(* CoDeSys 2.3 export: INDICATOR_CTRL.EXP *)

(* POU lib/INDICATOR_CTRL, FBD *)
FUNCTION_BLOCK INDICATOR_CTRL
VAR_INPUT
	iSTATE						:	INT;
	xEMERGENCY			:	BOOL;
	xRUNNING				:	BOOL;
	xCLOCK					:	BOOL;
END_VAR
VAR_OUTPUT
	_xIND_EMERGENCY			:	BOOL;
	_xIND_INIT_POS				:	BOOL;
	_xIND_PB_START			:	BOOL;
END_VAR
VAR
	xInitPos		:	BOOL;
END_VAR
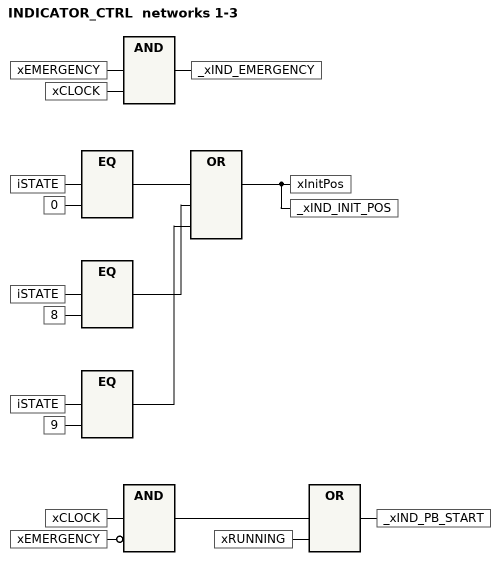
_FBD_ (* Function Block Diagram *)
NETWORK 1 (* Reset button should blink in case of emergency, indicating that a reset is needed. *)
	AND(xEMERGENCY, xCLOCK) => _xIND_EMERGENCY
NETWORK 2 (* The machine is in its initial position in state 0 (ready for start), state 8 (waiting for part to be picked up) or state 9 (resetting to state 0). *)
	<OR(EQ(iSTATE, 0), EQ(iSTATE, 8), EQ(iSTATE, 9)) => xInitPos> => _xIND_INIT_POS
NETWORK 3 (* PB should blink if emergency isn't engaged and the procution line isn't running and should light up permanently if it is running. *)
	OR(AND(xCLOCK, NOT xEMERGENCY), xRUNNING) => _xIND_PB_START
_END_FBD_
(* the same logic as Structured Text *)
(* Network 1: Reset button should blink in case of emergency, indicating that a reset is needed. *)
_xIND_EMERGENCY := xEMERGENCY AND xCLOCK;
(* Network 2: The machine is in its initial position in state 0 (ready for start), state 8 (waiting for part to be picked up) or state 9 (resetting to state 0). *)
xInitPos := (iSTATE = 0) OR (iSTATE = 8) OR (iSTATE = 9);
_xIND_INIT_POS := xInitPos;
(* Network 3: PB should blink if emergency isn't engaged and the procution line isn't running and should light up permanently if it is running. *)
_xIND_PB_START := (xCLOCK AND NOT xEMERGENCY) OR xRUNNING;
END_FUNCTION_BLOCK
